FUNCTION_BLOCK JobNotificationInterface (* Composite Function Block Type *)
  (* Standard: 61499-2 *)
  (* Version 0.0, 2018-03-05, 4DIAC-IDE, 4DIAC-Consortium *)
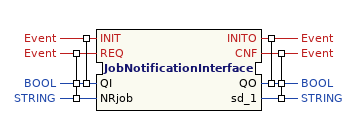
  EVENT_INPUT
    INIT WITH QI; (* Initialization Request *)
    REQ WITH QI, NRjob; (* Normal Execution Request *)
  END_EVENT
  EVENT_OUTPUT
    INITO WITH QO; (* Initialization Confirm *)
    CNF WITH QO, sd_1; (* Execution Confirmation *)
  END_EVENT
  VAR_INPUT
    QI : BOOL; (* Input event qualifier *)
    NRjob : STRING;
  END_VAR
  VAR_OUTPUT
    QO : BOOL; (* Output event qualifier *)
    sd_1 : STRING;
  END_VAR
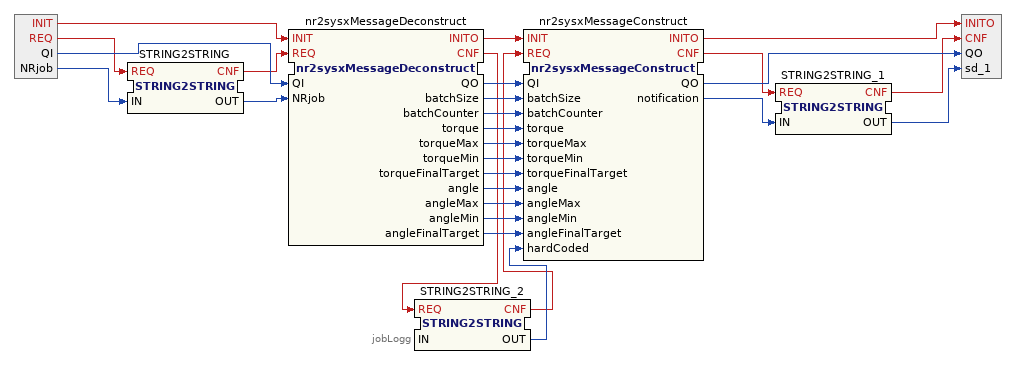
  FBS
    STRING2STRING : STRING2STRING;
    STRING2STRING_1 : STRING2STRING;
    STRING2STRING_2 : STRING2STRING(IN := jobLogg);
    nr2sysxMessageConstruct : nr2sysxMessageConstruct;
    nr2sysxMessageDeconstruct : nr2sysxMessageDeconstruct;
  END_FBS
  EVENT_CONNECTIONS
    REQ TO STRING2STRING.REQ;
    STRING2STRING.CNF TO nr2sysxMessageDeconstruct.REQ;
    INIT TO nr2sysxMessageDeconstruct.INIT;
    nr2sysxMessageDeconstruct.CNF TO STRING2STRING_2.REQ;
    nr2sysxMessageDeconstruct.INITO TO nr2sysxMessageConstruct.INIT;
    nr2sysxMessageConstruct.CNF TO STRING2STRING_1.REQ;
    STRING2STRING_1.CNF TO CNF;
    nr2sysxMessageConstruct.INITO TO INITO;
    STRING2STRING_2.CNF TO nr2sysxMessageConstruct.REQ;
  END_CONNECTIONS
  DATA_CONNECTIONS
    NRjob TO STRING2STRING.IN;
    STRING2STRING.OUT TO nr2sysxMessageDeconstruct.NRjob;
    QI TO nr2sysxMessageDeconstruct.QI;
    nr2sysxMessageDeconstruct.QO TO nr2sysxMessageConstruct.QI;
    nr2sysxMessageDeconstruct.batchSize TO nr2sysxMessageConstruct.batchSize;
    nr2sysxMessageDeconstruct.batchCounter TO nr2sysxMessageConstruct.batchCounter;
    nr2sysxMessageDeconstruct.torque TO nr2sysxMessageConstruct.torque;
    nr2sysxMessageDeconstruct.torqueMax TO nr2sysxMessageConstruct.torqueMax;
    nr2sysxMessageDeconstruct.torqueMin TO nr2sysxMessageConstruct.torqueMin;
    nr2sysxMessageDeconstruct.torqueFinalTarget TO nr2sysxMessageConstruct.torqueFinalTarget;
    nr2sysxMessageDeconstruct.angle TO nr2sysxMessageConstruct.angle;
    nr2sysxMessageDeconstruct.angleMax TO nr2sysxMessageConstruct.angleMax;
    nr2sysxMessageDeconstruct.angleMin TO nr2sysxMessageConstruct.angleMin;
    nr2sysxMessageDeconstruct.angleFinalTarget TO nr2sysxMessageConstruct.angleFinalTarget;
    STRING2STRING_2.OUT TO nr2sysxMessageConstruct.hardCoded;
    nr2sysxMessageConstruct.notification TO STRING2STRING_1.IN;
    STRING2STRING_1.OUT TO sd_1;
    nr2sysxMessageConstruct.QO TO QO;
  END_CONNECTIONS
END_FUNCTION_BLOCK
